# EPICS alarm handler configuration: devel/epics/apps/generalApp/alh/cryo.alhConfig
GROUP NULL CRYO
  $GUIDANCE
    For expert help on all cryogenic systems, page the engineering
    on-call person.
  $END
  CHANNEL CRYO B_cryotarget_LT_CR
    $GUIDANCE
      For MINOR (yellow) alarms please check that the cryo target He
      reservior is filling.  For MAJOR alarms please call the engineering
      on call number.
    $END
